FUNCTION TryConvert_BYTE_TO_ULINT : BOOL
VAR_INPUT
	in : BYTE;
	out : REFERENCE TO ULINT;
END_VAR

out := BYTE_TO_ULINT(in);
TryConvert_BYTE_TO_ULINT := TRUE;

END_FUNCTION

(* stored: Version 1.1.0.1, ProductVersion 3.1.4024.12
   POU TryConvert_BYTE_TO_ULINT: Id {2fc57219-1001-4d2f-b80b-59ab701b0ee0}, SpecialFunc None *)
